FUNCTION F_relu : LREAL
VAR_INPUT
	x : LREAL;
END_VAR

IF x<0 THEN
	F_relu := 0;
ELSE
	F_relu := x;	
END_IF

END_FUNCTION

(* stored: Version 1.1.0.1, ProductVersion 3.1.4024.12
   POU F_relu: Id {c25e9d73-e13f-4237-b9d6-69b1565e9352}, SpecialFunc None *)
